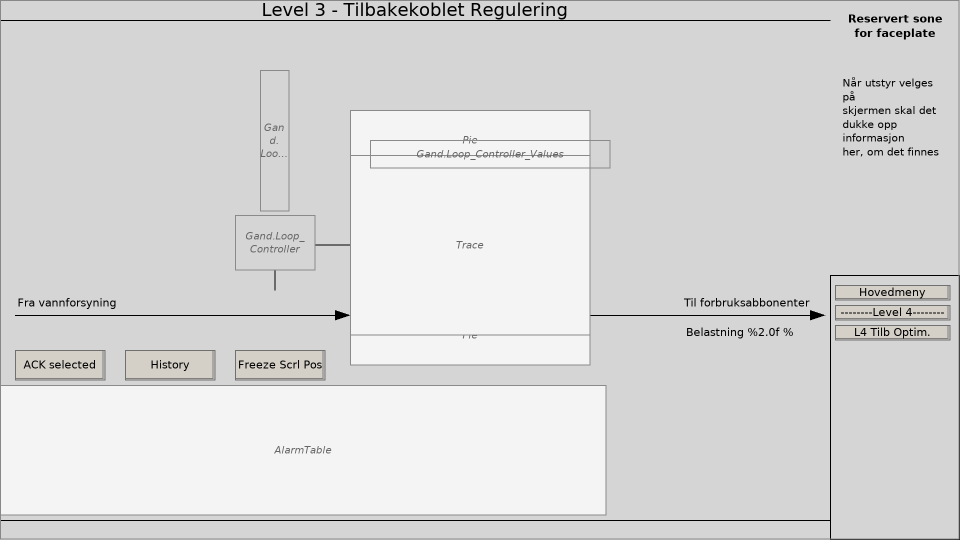
VISUALIZATION Level3_TilbakekobletRegulering  // 960x540
VAR_IN_OUT
END_VAR
VAR
	bResetTrigger : BOOL;
	bStart : BOOL;
	bStop : BOOL;
	bStore : BOOL;
	sStoreFilename : STRING;
	bRestore : BOOL;
	sRestoreFilename : STRING;
	bAckSel : BOOL;
	bHistory : BOOL;
	bFreezeScrlPos : BOOL;
END_VAR
    Rectangle (830,275 130x265)
    Frame (835,0 120x270)
        shows Faceplate_template()
        shows Navigation_template()
    Line (0,20) (830,20)
    Line (0,520) (830,520)
    Button (835,285 115x15), "Hovedmeny"
        OnMouseClick:  Assign=Hovedmeny, Type=Assignment
    Button (835,305 115x15), "--------Level 4--------"
        OnMouseClick:  Assign=Level4_TilbakekobletRegulering_Optimalisering, Type=Assignment
    Label (0,0 830x20), "Level 3 - Tilbakekoblet Regulering"
    Rectangle (350,140 240x195)
    Pie (350,110 240x60)
    Pie (350,305 240x60)
    Line (15,315) (335,315)
    Polygon (350,315) (335,310) (335,320)
    Line (590,315) (810,315)
    Polygon (825,315) (810,310) (810,320)
    Label (15,295 104x16), "Fra vannforsyning"
    Label (685,295 124x16), "Til forbruksabbonenter"
    Line (275,290) (275,270)
    Line (350,245) (315,245)
    Trace (350,155 240x180)
    Frame (235,215 80x55)
        shows Gand.Loop_Controller(Local_data := TilbakekobletRegulering.LOOP01)
    Frame (370,140 240x28)
        shows Gand.Loop_Controller_Values(Local_data := TilbakekobletRegulering.LOOP01)
    Textfield (665,320 150x25), "Belastning %2.0f %", text variable: TilbakekobletRegulering.Belastning_LIC01
        OnMouseClick: write the text variable via Default, min 0, max 100
    Frame (260,70 29x141)
        shows Gand.Loop_ControllerBar(Local_data := TilbakekobletRegulering.LOOP01)
    Button (835,325 115x15), "L4 Tilb Optim."
        OnMouseClick:  Assign=Level4_TilbakekobletRegulering_Optimalisering, Type=Assignment
    AlarmTable (0,385 606x130)
        p1521930926: __All
        p1663851261: __All
        p428520879: bAckSel
        p3266827225: bHistory
        p3894972949: bFreezeScrlPos
    Button (15,350 90x30), "ACK selected"
        toggle bAckSel
    Button (125,350 90x30), "History"
        toggle bHistory
    Button (235,350 90x30), "Freeze Scrl Pos"
        toggle bFreezeScrlPos
END_VISUALIZATION

(* text list AlarmGroup1 (id | default)
  0 | Nivå høyt i vanntank
   |  *)
